INTERFACE I_ChunkedResponseManager

METHOD PUBLIC HandleSuccessWithPayload;
VAR_INPUT
	OriginalResponse : I_ServerResponse;
	SourceAddress : PVOID;
	SourceSize : UDINT;
END_VAR
END_METHOD

METHOD PUBLIC TryHandleIncomingRequest : BOOL
VAR_INPUT
	Request : I_Request;
	Response : I_ServerResponse;
END_VAR
END_METHOD

END_INTERFACE

(* stored: Version 1.1.0.1, ProductVersion 3.1.4026.13
   Itf I_ChunkedResponseManager: Id {742749ff-d5f1-401d-ba14-a89597602dc3}
   Method HandleSuccessWithPayload: Id {cb9ed623-b3a3-4a92-9942-886b216880f9}
   Method TryHandleIncomingRequest: Id {004a329a-473d-4581-b23c-92ba35e334a3} *)
